TEXTLIST TextList_Config_Pompage
  0 = 'Conf pomp chambre' | FR: 'Pompage chambre' | EN: 'Chamber pumping'
  1 = 'Conf pomp sas' | FR: 'Pompage sas' | EN: 'Loadlock pumping'
  2 = 'TGF' | FR: 'Seuil de détection de grosse fuite' | EN: 'Gross leak detection threshold'
  3 = 'TGF delay' | FR: 'Temps de détection grosse fuite' | EN: 'Gross leak detection time'
  4 = 'ATM' | FR: 'Seuil de pression atmosphérique' | EN: 'Atmospheric pressure threshold'
  5 = 'Surventil' | FR: 'Temps de surventilation' | EN: 'Vent overtime'
  6 = 'PPrim' | FR: 'Seuil de basculement en pompage secondaire' | EN: 'High vacuum pumping start threshold'
  7 = 'RP PPrim' | FR: 'Seuil de détection de remontée de pression' | EN: 'Pressure rise detection threshold'
  8 = 'pprim delay' | FR: 'Temps de surveillance pompage primaire' | EN: 'Rough pumping monitoring time'
  9 = 'vent delay' | FR: 'Temps de surveillance ventilation' | EN: 'Venting monitoring time'
  10 = 'prm_pr_canon_ok' | FR: "Seuil d'autorisation allumage canon à électrons" | EN: 'E-gun starting authorization threshold'
  11 = 'prm_pr_canon_ion_ok' | FR: "Seuil d'autorisation allumage canon à ions" | EN: 'Ion gun starting authorization threshold'
  12 = 'PRM_tps_att_chaud' | FR: 'Temps de thermalisation' | EN: 'Thermalisation time'
  13 = 'Conf_Temp_Min' | FR: 'Température min. groupe chaud' | EN: 'Chiller minimum temperature'
  14 = 'Conf_Temp_Max' | FR: 'Température max. groupe chaud' | EN: 'Chiller maximum temperature'
  15 = 'vanne asservie' | FR: 'Vanne asservie' | EN: 'Servovalve'
  16 = 'Estimation du temps de pompage' | FR: 'Estimation du temps de pompage' | EN: 'Estimated pumping time'
  17 = 'Pump sweep time on pump balast / intersteel pump alternation' | FR: 'Temps balayage pompe sur alternance avec pompage interjoint' | EN: 'Pump sweep time on pump balast / intersteel pump alternation'
  18 = 'Intersteel pumping time on pump balast / intersteel pump alternation' | FR: 'Temps pompage interjoint sur alternance avec balayage pompe' | EN: 'Intersteel pumping time on pump balast / intersteel pump alternation'
  19 = 'Pump balast time before pump stop' | FR: 'Temps balayage pompe avant arrêt pompe' | EN: 'Pump balast time before pump stop'
  20 = 'Primary pump balast' | FR: 'Balayage pompe primaire' | EN: 'Primary pump balast'
   = ''
END_TEXTLIST

(* stored: Version 1.1.0.1, ProductVersion 3.1.4024.12
   TextList TextList_Config_Pompage: Id {c45795f6-a14a-4775-b20d-91a219b3b3c7} *)
